// TIA Portal project "PortaGaragemV002" (V14)
// O sistema de controle da porta deve abrir e
//  fechar a porta por meio de um painel de botões e
//  fornecer recursosde segurançapara evitaracidentes.

(* hardware
DEVICE "S7-1200 station_1"  S7-1200 Station
   slot 0: "Rack_0"  S7-1200 Rack  Rack  V1.0
   slot 1: "PLC_1"  CPU 1214C DC/DC/DC  6ES7 214-1AG40-0XB0  V4.2
*)

// ===== PLC "PLC_1"  CPU 1214C DC/DC/DC =====

VAR_GLOBAL   // PLC tag table "Default tag table"
   "System_Byte" AT %MB1 : Byte;
   "FirstScan" AT %M1.0 : Bool;
   "DiagStatusUpdate" AT %M1.1 : Bool;
   "AlwaysTRUE" AT %M1.2 : Bool;
   "AlwaysFALSE" AT %M1.3 : Bool;
   "Clock_Byte" AT %MB0 : Byte;
   "Clock_10Hz" AT %M0.0 : Bool;
   "Clock_5Hz" AT %M0.1 : Bool;
   "Clock_2.5Hz" AT %M0.2 : Bool;
   "Clock_2Hz" AT %M0.3 : Bool;
   "Clock_1.25Hz" AT %M0.4 : Bool;
   "Clock_1Hz" AT %M0.5 : Bool;
   "Clock_0.625Hz" AT %M0.6 : Bool;
   "Clock_0.5Hz" AT %M0.7 : Bool;
   "BotaoAbrir" AT %I0.1 : Bool;
   "BotaoFechar" AT %I0.2 : Bool;
   "SensorPortaAberta" AT %I0.3 : Bool;
   "SensorPortaFechada" AT %I0.4 : Bool;
   "SensorInfravermelhoSeg" AT %I0.5 : Bool;
   "MotorAbrePortao" AT %Q0.1 : Bool;
   "MotorFechaPortao" AT %Q0.2 : Bool;
END_VAR

FUNCTION "ControlePortao" : Void   // FC1, LAD
{ S7_Optimized_Access := 'TRUE' }
VERSION : 0.1
BEGIN

REGION Network 1: Comando Abrir Portao
   // Pressionar Botão_Abrir abre a porta, desde que não esteja aberta.
   //  A porta para de abrir quando o Sensor_Porta_Aberta é acionado.
   // Se o Feixe_Segurança detectar um objeto, a porta para de se mover.
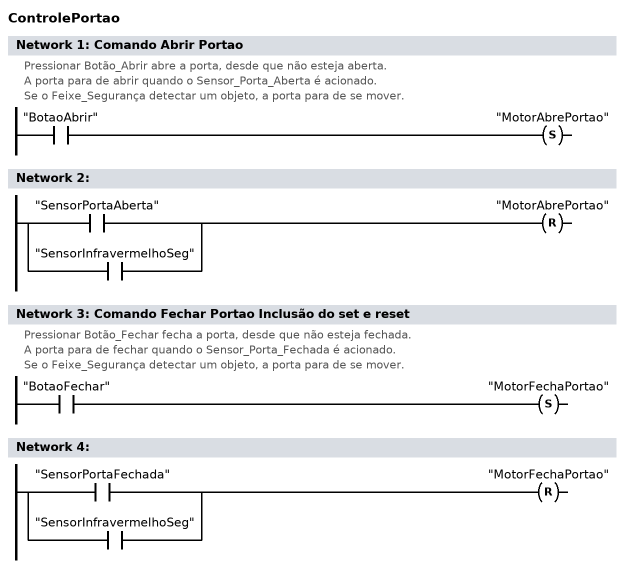
   RUNG wire#powerrail
      Contact( "BotaoAbrir" )
      S_Coil( "MotorAbrePortao" )
   END_RUNG
   // the same network as SCL:
   IF "BotaoAbrir" THEN "MotorAbrePortao" := TRUE; END_IF;
END_REGION

REGION Network 2
   RUNG wire#powerrail
      Contact( "SensorPortaAberta" )
      wire#w1
      R_Coil( "MotorAbrePortao" )
   END_RUNG
   RUNG wire#powerrail
      Contact( "SensorInfravermelhoSeg" )
   END_RUNG wire#w1
   // the same network as SCL:
   IF "SensorPortaAberta" OR "SensorInfravermelhoSeg" THEN "MotorAbrePortao" := FALSE; END_IF;
END_REGION

REGION Network 3: Comando Fechar Portao Inclusão do set e reset
   // Pressionar Botão_Fechar fecha a porta, desde que não esteja fechada.
   // A porta para de fechar quando o Sensor_Porta_Fechada é acionado.
   // Se o Feixe_Segurança detectar um objeto, a porta para de se mover.
   RUNG wire#powerrail
      Contact( "BotaoFechar" )
      S_Coil( "MotorFechaPortao" )
   END_RUNG
   // the same network as SCL:
   IF "BotaoFechar" THEN "MotorFechaPortao" := TRUE; END_IF;
END_REGION

REGION Network 4
   RUNG wire#powerrail
      Contact( "SensorPortaFechada" )
      wire#w1
      R_Coil( "MotorFechaPortao" )
   END_RUNG
   RUNG wire#powerrail
      Contact( "SensorInfravermelhoSeg" )
   END_RUNG wire#w1
   // the same network as SCL:
   IF "SensorPortaFechada" OR "SensorInfravermelhoSeg" THEN "MotorFechaPortao" := FALSE; END_IF;
END_REGION
END_FUNCTION

ORGANIZATION_BLOCK "Main"   // OB1, LAD, ProgramCycle
TITLE = "Main Program Sweep (Cycle)"
{ S7_Optimized_Access := 'TRUE' }
VERSION : 0.1
   VAR_INPUT
      Initial_Call : Bool;   // Initial call of this OB
      Remanence : Bool;   // =True, if remanent data are available
   END_VAR
BEGIN

REGION Network 1
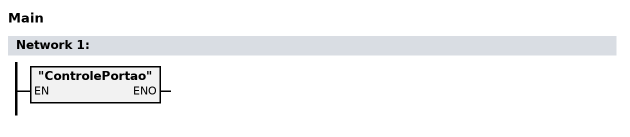
   RUNG wire#powerrail
      "ControlePortao"()
   END_RUNG
   // the same network as SCL:
   "ControlePortao"();
END_REGION
END_ORGANIZATION_BLOCK